DATA_BLOCK "ACTH"
{ S7_Optimized_Access := 'FALSE' }
VERSION : 0.1
NON_RETAIN
   STRUCT
      LAB10_AA001 : "VLVS_HMI";   // Регулятор рівня в барабані (Живильний клапан)
      HAD10_AA101 : "VLVS_HMI";   // Клапан неперевної продувки
      LBA10_AA102 : "VLVD_HMI";   // ГПЗ
      SGA20_AA601 : "VLVD_HMI";   // Клапан пожежогасіння транспортера №1
      SGA20_AA602 : "VLVD_HMI";   // Клапан пожежогасіння транспортера №2
      EBA10_AA101 : "VLVD_HMI";   // Відсічний затвор №1 бункеру палива
      EBA20_AA102 : "VLVD_HMI";   // Відсічний затвор №2 бункеру палива
      HLA10_AA151 : "VLVD_HMI";   // Шибер первинного повітря №1
      HLA10_AA152 : "VLVD_HMI";   // Шибер первинного повітря №2
      HHB11_P001 : "VLVD_HMI";   // Колосникова решітка. Поле №1
      HHB12_P002 : "VLVD_HMI";   // Колосникова решітка. Поле №2
      HHB13_P003 : "VLVD_HMI";   // Колосникова решітка. Поле №3
      HHB14_P004 : "VLVD_HMI";   // Колосникова решітка. Поле №4
      LAB01_AP001 : "DRVS_HMI";   // Живильний насос №1
      LAB02_AP002 : "DRVS_HMI";   // Живильний насос №2
      HFB11_AF001 : "DRVS_HMI";   // Шнек подачі палива №1
      HFB21_AF001 : "DRVS_HMI";   // Шнек подачі палива №2
      HFB12_AF001 : "DRVS_HMI";   // Транспортер подачі палива №1
      HFB22_AF001 : "DRVS_HMI";   // Транспортер подачі палива №2
      EKG11_AF001 : "DRVS_HMI";   // Пульсатор
      HLA10_AF001 : "DRVS_HMI";   // Вентилятор первинного дуття ДВ1
      HLA20_AF001 : "DRVS_HMI";   // Вентилятор вторинного дуття ДВ2
      HNC10_AF001 : "DRVS_HMI";   // Димосос ДН1
      HNC20_AF001 : "DRVS_HMI";   // Димосос ДН2
      Rez1 : "DRVS_HMI";   // Резервний привод ПЧ
      Rez2 : "DRVD_HMI";   // Резервний привод №2
      EKG10_AN001 : "DRVD_HMI";   // Вентилятор закиду палива ВЛ
      ETC10_AF001 : "DRVD_HMI";   // Конвеєр золи скребковий №1
      ETC01_AF001 : "DRVD_HMI";   // Конвеєр золи скребковий №2
      ETC01_AF002 : "DRVD_HMI";   // Конвеєр золи гвинтовий №3
      ETG21_AF001 : "DRVD_HMI";   // Шлюзовий затвор №1 (з під 1 колос. решітки)
      ETG22_AF001 : "DRVD_HMI";   // Шлюзовий затвор №2 (з під 2 колос. решітки)
      ETG23_AF001 : "DRVD_HMI";   // Шлюзовий затвор №3 (з під 3 колос. решітки)
      ETG24_AF001 : "DRVD_HMI";   // Шлюзовий затвор №4 (з під 4 колос. решітки)
      ETG31_AF001 : "DRVD_HMI";   // Шлюзовий затвор №5 (з під 1 конвект. частини)
      ETG32_AF001 : "DRVD_HMI";   // Шлюзовий затвор №6 (з під 2 конвект. частини)
      ETG41_AF001 : "DRVD_HMI";   // Шлюзовий затвор №7 (з під економайзера)
      ETG51_AF001 : "DRVD_HMI";   // Шлюзовий затвор №8 (з під циклона)
      ETG31_AF002 : "DRVD_HMI";   // Шнек золовидалення №1 (з під 1 конвект. частини)
      ETG32_AF002 : "DRVD_HMI";   // Шнек золовидалення №2 (з під 2 конвект. частини)
      ETG51_AF002 : "DRVD_HMI";   // Шнек золовидалення №3 (з під циклона)
      HCB10_AN001 : "DRVD_HMI";   // Обдувочний апарат №1
      HCB20_AN001 : "DRVD_HMI";   // Обдувочний апарат №2
      HCB30_AN001 : "DRVD_HMI";   // Обдувочний апарат №3
      HCB40_AN001 : "DRVD_HMI";   // Обдувочний апарат №4
      HCB50_AN001 : "DRVD_HMI";   // Обдувочний апарат №5
      HCB60_AN001 : "DRVD_HMI";   // Обдувочний апарат №6
      HCB70_AN001 : "DRVD_HMI";   // Обдувочний апарат №7
      HCB80_AN001 : "DRVD_HMI";   // Обдувочний апарат №8
      HCB90_AN001 : "DRVD_HMI";   // Обдувочний апарат №9
      HCB100_AN001 : "DRVD_HMI";   // Обдувочний апарат №10
      HCB100_AN002 : "VLVD_HMI";   // Каретка Обдувочного апарату №10
      HCB10_AA601 : "VLVD_HMI";   // Клапан Обдувного апарату №1
      HCB20_AA601 : "VLVD_HMI";   // Клапан Обдувного апарату №2
      HCB30_AA601 : "VLVD_HMI";   // Клапан Обдувного апарату №3
      HCB40_AA601 : "VLVD_HMI";   // Клапан Обдувного апарату №4
      HCB50_AA601 : "VLVD_HMI";   // Клапан Обдувного апарату №5
      HCB60_AA601 : "VLVD_HMI";   // Клапан Обдувного апарату №6
      HCB70_AA601 : "VLVD_HMI";   // Клапан Обдувного апарату №7
      HCB80_AA601 : "VLVD_HMI";   // Клапан Обдувного апарату №8
      HCB90_AA601 : "VLVD_HMI";   // Клапан Обдувного апарату №9
      HCB100_AA601 : "VLVD_HMI";   // Клапан Обдувного апарату №10
   END_STRUCT;


BEGIN

END_DATA_BLOCK

